FUNCTION_BLOCK FB_SkillBasis
VAR_INPUT
	
END_VAR
VAR_OUTPUT
END_VAR
VAR
	// Interne Variablen
	bStart					:BOOL;
	bStop					:BOOL;
	
	// SFC-Flags
	SFCReset				:BOOL;
END_VAR

METHOD M_Reset : BOOL
VAR_INPUT
END_VAR
bStart := FALSE;
bStop := FALSE; 
SFCReset := TRUE;
END_METHOD

METHOD M_Start : BOOL
VAR_INPUT
END_VAR
SFCReset := FALSE;
bStop := FALSE;
bStart := TRUE;
END_METHOD

METHOD M_Stop : BOOL
VAR_INPUT
END_VAR
bStart := FALSE; 
bStop := TRUE;
END_METHOD

PROPERTY P_Finished : BOOL
GET
P_Finished := bStop;
END_GET
END_PROPERTY

END_FUNCTION_BLOCK

(* stored: Version 1.1.0.1
   POU FB_SkillBasis: Id {f9e67a08-8c82-42a7-bd97-06b217ca57b3}, SpecialFunc None
   Method M_Reset: Id {20f226ac-830d-4f12-9db0-d8115b45c003}
   Method M_Start: Id {0a0d5daf-819b-444a-a481-e231b0a4e151}
   Method M_Stop: Id {fa44c262-cbc9-425f-a719-318e4bb27629}
   Property P_Finished: Id {7064e54d-7363-4993-b3da-29f36e7f79fb}
   Get Get: Id {39d70dfe-e51c-4fd8-8d9f-2e82f9b63d0b} *)
